{attribute addProperty BoxType "KL6211-0020"}
{attribute addProperty Id "Channel_1Channel_B94E0A4200"}
{attribute addProperty CRC "4077508386"}
{attribute addProperty SizeInBites "0"}
{attribute addProperty SizeInBytes "0"}
TYPE KL_F309D722 :
STRUCT
	{attribute addProperty Name "Channel_1"}
	Channel_1 : Channel_B94E0A42;
END_STRUCT
END_TYPE

(* stored: Version 1.2.0.0, ProductVersion 3.1.4024.9
   DUT KL_F309D722: Id {88b9e9a5-5f70-4bc5-9392-4ad8859f27fb} *)
